//=============================================================================
// ST10_Flow14_B2Press.scl
// 1:1 CONVERSION FROM TIA PORTAL V18 GRAPH XML
// Generated: 2026-02-02
//=============================================================================

TYPE
    E_STEP_ST10_Flow14_B2Press : (
        STEP_ST10_Flow14_B2Press_S2 := 2,
        STEP_ST10_Flow14_B2Press_MesCheckResult_1 := 309,
        STEP_ST10_Flow14_B2Press_ResultOKData := 145,
        STEP_ST10_Flow14_B2Press_B_PressFitting_01CylinderToHP_1 := 140,
        STEP_ST10_Flow14_B2Press_Process_FInish := 237,
        STEP_ST10_Flow14_B2Press_ShaftAndRingOK := 16,
        STEP_ST10_Flow14_B2Press_PutRing := 127,
        STEP_ST10_Flow14_B2Press_PressProgram_1 := 20,
        STEP_ST10_Flow14_B2Press_MESOK := 19,
        STEP_ST10_Flow14_B2Press_Wait_robot_finish_task := 131,
        STEP_ST10_Flow14_B2Press_Step15 := 24,
        STEP_ST10_Flow14_B2Press_Wait__robot_finish_task_1 := 134,
        STEP_ST10_Flow14_B2Press_Status_Alarm := 118,
        STEP_ST10_Flow14_B2Press_StartCycle := 141,
        STEP_ST10_Flow14_B2Press_PressProgram := 8,
        STEP_ST10_Flow14_B2Press_Step400 := 400,
        STEP_ST10_Flow14_B2Press_NGCount := 404,
        STEP_ST10_Flow14_B2Press_RobotLeavePress_Area := 115,
        STEP_ST10_Flow14_B2Press_Part_Check := 239,
        STEP_ST10_Flow14_B2Press_Bypass := 316,
        STEP_ST10_Flow14_B2Press_PartStatus_1 := 137,
        STEP_ST10_Flow14_B2Press_B_PressFitting_01GripperCylinderToHP := 116,
        STEP_ST10_Flow14_B2Press_Bypass_1 := 319,
        STEP_ST10_Flow14_B2Press_Wait_robot_in_safety_area := 133,
        STEP_ST10_Flow14_B2Press_Request_robot_putShaft := 112,
        STEP_ST10_Flow14_B2Press_Prepare_MES_CheckData := 305,
        STEP_ST10_Flow14_B2Press_MesCheckIn_1 := 314,
        STEP_ST10_Flow14_B2Press_PartCheck := 238,
        STEP_ST10_Flow14_B2Press_Step313 := 317,
        STEP_ST10_Flow14_B2Press_Pressing := 200,
        STEP_ST10_Flow14_B2Press_Request_robot_pick := 408,
        STEP_ST10_Flow14_B2Press_ProcessStart := 100,
        STEP_ST10_Flow14_B2Press_MES := 18,
        STEP_ST10_Flow14_B2Press_CheckPressGripStatus := 15,
        STEP_ST10_Flow14_B2Press_MES_1NG := 25,
        STEP_ST10_Flow14_B2Press_CheckPressSensor := 138,
        STEP_ST10_Flow14_B2Press_PressHoming := 9,
        STEP_ST10_Flow14_B2Press_F14_Initial := 1,
        STEP_ST10_Flow14_B2Press_DataMove := 132,
        STEP_ST10_Flow14_B2Press_MES_Check_NG_3 := 318,
        STEP_ST10_Flow14_B2Press_MESOverTime_1 := 312,
        STEP_ST10_Flow14_B2Press_ProcessFInish_1 := 143,
        STEP_ST10_Flow14_B2Press_ShaftOK := 125,
        STEP_ST10_Flow14_B2Press_ProcessFinish := 403,
        STEP_ST10_Flow14_B2Press_PressHoming_1 := 21,
        STEP_ST10_Flow14_B2Press_ResetMesCheckRequest := 301,
        STEP_ST10_Flow14_B2Press_B_PressFitting_01CylinderToHP := 120,
        STEP_ST10_Flow14_B2Press_CheckPressProgram := 139,
        STEP_ST10_Flow14_B2Press_CheckPressResult := 144,
        STEP_ST10_Flow14_B2Press_OKCount := 402,
        STEP_ST10_Flow14_B2Press_PressHoming_ := 13,
        STEP_ST10_Flow14_B2Press_MES_Result := 500,
        STEP_ST10_Flow14_B2Press_ProcessFinsh := 605,
        STEP_ST10_Flow14_B2Press_Request_robot_putRing := 113,
        STEP_ST10_Flow14_B2Press_MES_Check_Finish := 515,
        STEP_ST10_Flow14_B2Press_WaitPressFinish := 201,
        STEP_ST10_Flow14_B2Press_S3 := 3,
        STEP_ST10_Flow14_B2Press_CheckFinish_1 := 315,
        STEP_ST10_Flow14_B2Press_PressReady__1 := 22,
        STEP_ST10_Flow14_B2Press_B_PressFitting_01GripperCylinderToWP := 119,
        STEP_ST10_Flow14_B2Press_DataClear := 604,
        STEP_ST10_Flow14_B2Press_Step314 := 320,
        STEP_ST10_Flow14_B2Press_MES_Check_NG_2 := 313,
        STEP_ST10_Flow14_B2Press_ProductCheckAlarm := 240,
        STEP_ST10_Flow14_B2Press_CheckRingExist := 117,
        STEP_ST10_Flow14_B2Press_ProcessStart_CTStart := 104,
        STEP_ST10_Flow14_B2Press_RobotPick := 600,
        STEP_ST10_Flow14_B2Press_ResetMesUnloadRequest_1 := 302,
        STEP_ST10_Flow14_B2Press_CheckPressReady := 208,
        STEP_ST10_Flow14_B2Press_ProductCheckAlarm_1 := 241,
        STEP_ST10_Flow14_B2Press_StatusAlarm := 126,
        STEP_ST10_Flow14_B2Press_ResultNGData := 146,
        STEP_ST10_Flow14_B2Press_MESOverTime := 321,
        STEP_ST10_Flow14_B2Press_JudgeStatus := 401,
        STEP_ST10_Flow14_B2Press_PressHoming__1 := 23,
        STEP_ST10_Flow14_B2Press_PressReady_ := 12,
        STEP_ST10_Flow14_B2Press_Prepare_MES_CheckData_1 := 307,
        STEP_ST10_Flow14_B2Press_Normal_mode := 103,
        STEP_ST10_Flow14_B2Press_Step147 := 147,
        STEP_ST10_Flow14_B2Press_S5_MESInitial := 5,
        STEP_ST10_Flow14_B2Press_NoPart := 129,
        STEP_ST10_Flow14_B2Press_Wait__robot_finish_task := 130,
        STEP_ST10_Flow14_B2Press_PartStatus := 123,
        STEP_ST10_Flow14_B2Press_Press_NG := 17,
        STEP_ST10_Flow14_B2Press_CheckMachineStatus := 102,
        STEP_ST10_Flow14_B2Press_ok_1 := 322,
        STEP_ST10_Flow14_B2Press_Step14 := 14,
        STEP_ST10_Flow14_B2Press_Determine_product_status := 101,
        STEP_ST10_Flow14_B2Press_MES_Result_OK_1 := 405,
        STEP_ST10_Flow14_B2Press_MES__Check___In := 150,
        STEP_ST10_Flow14_B2Press_RobotLeavePressArea := 121,
        STEP_ST10_Flow14_B2Press_S10_InitialFinish := 10,
        STEP_ST10_Flow14_B2Press_S4 := 4,
        STEP_ST10_Flow14_B2Press_ResetPressStart := 142,
    ) INT := 1;
END_TYPE

CONST
    STEP_ST10_Flow14_B2Press_S2 := 2;
    STEP_ST10_Flow14_B2Press_MesCheckResult_1 := 309;
    STEP_ST10_Flow14_B2Press_ResultOKData := 145;
    STEP_ST10_Flow14_B2Press_B_PressFitting_01CylinderToHP_1 := 140;
    STEP_ST10_Flow14_B2Press_Process_FInish := 237;
    STEP_ST10_Flow14_B2Press_ShaftAndRingOK := 16;
    STEP_ST10_Flow14_B2Press_PutRing := 127;
    STEP_ST10_Flow14_B2Press_PressProgram_1 := 20;
    STEP_ST10_Flow14_B2Press_MESOK := 19;
    STEP_ST10_Flow14_B2Press_Wait_robot_finish_task := 131;
    STEP_ST10_Flow14_B2Press_Step15 := 24;
    STEP_ST10_Flow14_B2Press_Wait__robot_finish_task_1 := 134;
    STEP_ST10_Flow14_B2Press_Status_Alarm := 118;
    STEP_ST10_Flow14_B2Press_StartCycle := 141;
    STEP_ST10_Flow14_B2Press_PressProgram := 8;
    STEP_ST10_Flow14_B2Press_Step400 := 400;
    STEP_ST10_Flow14_B2Press_NGCount := 404;
    STEP_ST10_Flow14_B2Press_RobotLeavePress_Area := 115;
    STEP_ST10_Flow14_B2Press_Part_Check := 239;
    STEP_ST10_Flow14_B2Press_Bypass := 316;
    STEP_ST10_Flow14_B2Press_PartStatus_1 := 137;
    STEP_ST10_Flow14_B2Press_B_PressFitting_01GripperCylinderToHP := 116;
    STEP_ST10_Flow14_B2Press_Bypass_1 := 319;
    STEP_ST10_Flow14_B2Press_Wait_robot_in_safety_area := 133;
    STEP_ST10_Flow14_B2Press_Request_robot_putShaft := 112;
    STEP_ST10_Flow14_B2Press_Prepare_MES_CheckData := 305;
    STEP_ST10_Flow14_B2Press_MesCheckIn_1 := 314;
    STEP_ST10_Flow14_B2Press_PartCheck := 238;
    STEP_ST10_Flow14_B2Press_Step313 := 317;
    STEP_ST10_Flow14_B2Press_Pressing := 200;
    STEP_ST10_Flow14_B2Press_Request_robot_pick := 408;
    STEP_ST10_Flow14_B2Press_ProcessStart := 100;
    STEP_ST10_Flow14_B2Press_MES := 18;
    STEP_ST10_Flow14_B2Press_CheckPressGripStatus := 15;
    STEP_ST10_Flow14_B2Press_MES_1NG := 25;
    STEP_ST10_Flow14_B2Press_CheckPressSensor := 138;
    STEP_ST10_Flow14_B2Press_PressHoming := 9;
    STEP_ST10_Flow14_B2Press_F14_Initial := 1;
    STEP_ST10_Flow14_B2Press_DataMove := 132;
    STEP_ST10_Flow14_B2Press_MES_Check_NG_3 := 318;
    STEP_ST10_Flow14_B2Press_MESOverTime_1 := 312;
    STEP_ST10_Flow14_B2Press_ProcessFInish_1 := 143;
    STEP_ST10_Flow14_B2Press_ShaftOK := 125;
    STEP_ST10_Flow14_B2Press_ProcessFinish := 403;
    STEP_ST10_Flow14_B2Press_PressHoming_1 := 21;
    STEP_ST10_Flow14_B2Press_ResetMesCheckRequest := 301;
    STEP_ST10_Flow14_B2Press_B_PressFitting_01CylinderToHP := 120;
    STEP_ST10_Flow14_B2Press_CheckPressProgram := 139;
    STEP_ST10_Flow14_B2Press_CheckPressResult := 144;
    STEP_ST10_Flow14_B2Press_OKCount := 402;
    STEP_ST10_Flow14_B2Press_PressHoming_ := 13;
    STEP_ST10_Flow14_B2Press_MES_Result := 500;
    STEP_ST10_Flow14_B2Press_ProcessFinsh := 605;
    STEP_ST10_Flow14_B2Press_Request_robot_putRing := 113;
    STEP_ST10_Flow14_B2Press_MES_Check_Finish := 515;
    STEP_ST10_Flow14_B2Press_WaitPressFinish := 201;
    STEP_ST10_Flow14_B2Press_S3 := 3;
    STEP_ST10_Flow14_B2Press_CheckFinish_1 := 315;
    STEP_ST10_Flow14_B2Press_PressReady__1 := 22;
    STEP_ST10_Flow14_B2Press_B_PressFitting_01GripperCylinderToWP := 119;
    STEP_ST10_Flow14_B2Press_DataClear := 604;
    STEP_ST10_Flow14_B2Press_Step314 := 320;
    STEP_ST10_Flow14_B2Press_MES_Check_NG_2 := 313;
    STEP_ST10_Flow14_B2Press_ProductCheckAlarm := 240;
    STEP_ST10_Flow14_B2Press_CheckRingExist := 117;
    STEP_ST10_Flow14_B2Press_ProcessStart_CTStart := 104;
    STEP_ST10_Flow14_B2Press_RobotPick := 600;
    STEP_ST10_Flow14_B2Press_ResetMesUnloadRequest_1 := 302;
    STEP_ST10_Flow14_B2Press_CheckPressReady := 208;
    STEP_ST10_Flow14_B2Press_ProductCheckAlarm_1 := 241;
    STEP_ST10_Flow14_B2Press_StatusAlarm := 126;
    STEP_ST10_Flow14_B2Press_ResultNGData := 146;
    STEP_ST10_Flow14_B2Press_MESOverTime := 321;
    STEP_ST10_Flow14_B2Press_JudgeStatus := 401;
    STEP_ST10_Flow14_B2Press_PressHoming__1 := 23;
    STEP_ST10_Flow14_B2Press_PressReady_ := 12;
    STEP_ST10_Flow14_B2Press_Prepare_MES_CheckData_1 := 307;
    STEP_ST10_Flow14_B2Press_Normal_mode := 103;
    STEP_ST10_Flow14_B2Press_Step147 := 147;
    STEP_ST10_Flow14_B2Press_S5_MESInitial := 5;
    STEP_ST10_Flow14_B2Press_NoPart := 129;
    STEP_ST10_Flow14_B2Press_Wait__robot_finish_task := 130;
    STEP_ST10_Flow14_B2Press_PartStatus := 123;
    STEP_ST10_Flow14_B2Press_Press_NG := 17;
    STEP_ST10_Flow14_B2Press_CheckMachineStatus := 102;
    STEP_ST10_Flow14_B2Press_ok_1 := 322;
    STEP_ST10_Flow14_B2Press_Step14 := 14;
    STEP_ST10_Flow14_B2Press_Determine_product_status := 101;
    STEP_ST10_Flow14_B2Press_MES_Result_OK_1 := 405;
    STEP_ST10_Flow14_B2Press_MES__Check___In := 150;
    STEP_ST10_Flow14_B2Press_RobotLeavePressArea := 121;
    STEP_ST10_Flow14_B2Press_S10_InitialFinish := 10;
    STEP_ST10_Flow14_B2Press_S4 := 4;
    STEP_ST10_Flow14_B2Press_ResetPressStart := 142;
END_CONST

FUNCTION_BLOCK "ST10_Flow14_B2Press_1to1"
{ S7_Optimized_Access := 'TRUE' }
VERSION : 1.0

VAR_INPUT
    iSysInface : "RCS_SysComInterface_V1";
END_VAR

VAR_IN_OUT
    ioPM_Inface : "RCS_PMInterface_V1";
    ioStatus : Int;
END_VAR

VAR_OUTPUT
    oAlarmID : Int;
END_VAR

VAR
    State : INT := 1;
    act_InitialRun : Bool;
    act_InitialOK : Bool;
    act_WaitRunning : Bool;
    act_Running : Bool;
    act_ProcessComplete : Bool;
    act_ProcessStart : Bool;
    act_UnPause : Bool;
    bError : Bool;
    wErrorID : Word;
END_VAR

BEGIN
    //======================================================================
    // STATE MACHINE - Inline Transition Conditions
    //======================================================================

    CASE #State OF

        // ===========================================
        // STEP 2: S2
        // ===========================================
        STEP_ST10_Flow14_B2Press_S2:
            // No actions in XML

            // Transition to next step: 309
            IF TRUE THEN  // Sequential transition - review XML for actual condition
                #State := STEP_ST10_Flow14_B2Press_MesCheckResult_1;
            END_IF;

        // ===========================================
        // STEP 309: MesCheckResult_1
        // ===========================================
        STEP_ST10_Flow14_B2Press_MesCheckResult_1:
            // Action Qualifier=N
            // Token: "PLCtoMES"."PLC.Unload_Station7DataSaveReq"
            "PLCtoMES"."PLC.Unload_Station7DataSaveReq";

            // Transition to next step: 145
            IF TRUE THEN  // Sequential transition - review XML for actual condition
                #State := STEP_ST10_Flow14_B2Press_ResultOKData;
            END_IF;

        // ===========================================
        // STEP 145: ResultOKData
        // ===========================================
        STEP_ST10_Flow14_B2Press_ResultOKData:
            // Action Qualifier=N
            // Token: "AutoProcessData".B_Press2.PartStatus := 480
            "AutoProcessData".B_Press2.PartStatus := 480;

            // Transition to next step: 140
            IF TRUE THEN  // Sequential transition - review XML for actual condition
                #State := STEP_ST10_Flow14_B2Press_B_PressFitting_01CylinderToHP_1;
            END_IF;

        // ===========================================
        // STEP 140: B-PressFitting-01CylinderToHP_1
        // ===========================================
        STEP_ST10_Flow14_B2Press_B_PressFitting_01CylinderToHP_1:
            // Action Qualifier=S
            // Token: "ST10Cylinder".Cy[8].Inout.AutoGoHome
            "ST10Cylinder".Cy[8].Inout.AutoGoHome := TRUE;
            // Action Qualifier=R
            // Token: "ST10Cylinder".Cy[8].Inout.AutoGoWork
            "ST10Cylinder".Cy[8].Inout.AutoGoWork := FALSE;

            // Transition to next step: 237
            IF TRUE THEN  // Sequential transition - review XML for actual condition
                #State := STEP_ST10_Flow14_B2Press_Process_FInish;
            END_IF;

        // ===========================================
        // STEP 237: Process FInish
        // ===========================================
        STEP_ST10_Flow14_B2Press_Process_FInish:
            // No actions in XML

            // Transition to next step: 16
            IF TRUE THEN  // Sequential transition - review XML for actual condition
                #State := STEP_ST10_Flow14_B2Press_ShaftAndRingOK;
            END_IF;

        // ===========================================
        // STEP 16: ShaftAndRingOK
        // ===========================================
        STEP_ST10_Flow14_B2Press_ShaftAndRingOK:
            // No actions in XML

            // Transition to next step: 127
            IF TRUE THEN  // Sequential transition - review XML for actual condition
                #State := STEP_ST10_Flow14_B2Press_PutRing;
            END_IF;

        // ===========================================
        // STEP 127: PutRing
        // ===========================================
        STEP_ST10_Flow14_B2Press_PutRing:
            // No actions in XML

            // Transition to next step: 20
            IF TRUE THEN  // Sequential transition - review XML for actual condition
                #State := STEP_ST10_Flow14_B2Press_PressProgram_1;
            END_IF;

        // ===========================================
        // STEP 20: PressProgram_1
        // ===========================================
        STEP_ST10_Flow14_B2Press_PressProgram_1:
            // Action Qualifier=N
            // Token: "DB_maXYmosNC2".ProgNo := 1
            "DB_maXYmosNC2".ProgNo := 1;

            // Transition to next step: 19
            IF TRUE THEN  // Sequential transition - review XML for actual condition
                #State := STEP_ST10_Flow14_B2Press_MESOK;
            END_IF;

        // ===========================================
        // STEP 19: MESOK
        // ===========================================
        STEP_ST10_Flow14_B2Press_MESOK:
            // No actions in XML

            // Transition to next step: 131
            IF TRUE THEN  // Sequential transition - review XML for actual condition
                #State := STEP_ST10_Flow14_B2Press_Wait_robot_finish_task;
            END_IF;

        // ===========================================
        // STEP 131: Wait robot finish task
        // ===========================================
        STEP_ST10_Flow14_B2Press_Wait_robot_finish_task:
            // No actions in XML

            // Transition to next step: 24
            IF TRUE THEN  // Sequential transition - review XML for actual condition
                #State := STEP_ST10_Flow14_B2Press_Step15;
            END_IF;

        // ===========================================
        // STEP 24: Step15
        // ===========================================
        STEP_ST10_Flow14_B2Press_Step15:
            // No actions in XML

            // Transition to next step: 134
            IF TRUE THEN  // Sequential transition - review XML for actual condition
                #State := STEP_ST10_Flow14_B2Press_Wait__robot_finish_task_1;
            END_IF;

        // ===========================================
        // STEP 134: Wait  robot finish task_1
        // ===========================================
        STEP_ST10_Flow14_B2Press_Wait__robot_finish_task_1:
            // No actions in XML

            // Transition to next step: 118
            IF TRUE THEN  // Sequential transition - review XML for actual condition
                #State := STEP_ST10_Flow14_B2Press_Status_Alarm;
            END_IF;

        // ===========================================
        // STEP 118: Status Alarm
        // ===========================================
        STEP_ST10_Flow14_B2Press_Status_Alarm:
            // Action Qualifier=S
            // Token: "ST10_DeviceError".B.B2Press.StatusError
            "ST10_DeviceError".B.B2Press.StatusError := TRUE;

            // Transition to next step: 141
            IF TRUE THEN  // Sequential transition - review XML for actual condition
                #State := STEP_ST10_Flow14_B2Press_StartCycle;
            END_IF;

        // ===========================================
        // STEP 141: StartCycle
        // ===========================================
        STEP_ST10_Flow14_B2Press_StartCycle:
            // Action Qualifier=S
            // Token: "DB_maXYmosNC2".StartCycle
            "DB_maXYmosNC2".StartCycle := TRUE;

            // Transition to next step: 8
            IF TRUE THEN  // Sequential transition - review XML for actual condition
                #State := STEP_ST10_Flow14_B2Press_PressProgram;
            END_IF;

        // ===========================================
        // STEP 8: PressProgram
        // ===========================================
        STEP_ST10_Flow14_B2Press_PressProgram:
            // Action Qualifier=N
            // Token: "DB_maXYmosNC2".ProgNo := 1
            "DB_maXYmosNC2".ProgNo := 1;

            // Transition to next step: 400
            IF TRUE THEN  // Sequential transition - review XML for actual condition
                #State := STEP_ST10_Flow14_B2Press_Step400;
            END_IF;

        // ===========================================
        // STEP 400: Step400
        // ===========================================
        STEP_ST10_Flow14_B2Press_Step400:
            // No actions in XML

            // Transition to next step: 404
            IF TRUE THEN  // Sequential transition - review XML for actual condition
                #State := STEP_ST10_Flow14_B2Press_NGCount;
            END_IF;

        // ===========================================
        // STEP 404: NGCount
        // ===========================================
        STEP_ST10_Flow14_B2Press_NGCount:
            // Action Qualifier=N
            // Token: #ioPM_Inface.ProcessResult := #ioStatus
            #ioPM_Inface.ProcessResult := #ioStatus;

            // Transition to next step: 115
            IF TRUE THEN  // Sequential transition - review XML for actual condition
                #State := STEP_ST10_Flow14_B2Press_RobotLeavePress_Area;
            END_IF;

        // ===========================================
        // STEP 115: RobotLeavePress Area
        // ===========================================
        STEP_ST10_Flow14_B2Press_RobotLeavePress_Area:
            // No actions in XML

            // Transition to next step: 239
            IF TRUE THEN  // Sequential transition - review XML for actual condition
                #State := STEP_ST10_Flow14_B2Press_Part_Check;
            END_IF;

        // ===========================================
        // STEP 239: Part Check
        // ===========================================
        STEP_ST10_Flow14_B2Press_Part_Check:
            // No actions in XML

            // Transition to next step: 316
            IF TRUE THEN  // Sequential transition - review XML for actual condition
                #State := STEP_ST10_Flow14_B2Press_Bypass;
            END_IF;

        // ===========================================
        // STEP 316: Bypass
        // ===========================================
        STEP_ST10_Flow14_B2Press_Bypass:
            // No actions in XML

            // Transition to next step: 137
            IF TRUE THEN  // Sequential transition - review XML for actual condition
                #State := STEP_ST10_Flow14_B2Press_PartStatus_1;
            END_IF;

        // ===========================================
        // STEP 137: PartStatus_1
        // ===========================================
        STEP_ST10_Flow14_B2Press_PartStatus_1:
            // Action Qualifier=N
            // Token: "AutoProcessData".B_Press2.PartStatus := 450
            "AutoProcessData".B_Press2.PartStatus := 450;

            // Transition to next step: 116
            IF TRUE THEN  // Sequential transition - review XML for actual condition
                #State := STEP_ST10_Flow14_B2Press_B_PressFitting_01GripperCylinderToHP;
            END_IF;

        // ===========================================
        // STEP 116: B-PressFitting-01GripperCylinderToHP
        // ===========================================
        STEP_ST10_Flow14_B2Press_B_PressFitting_01GripperCylinderToHP:
            // Action Qualifier=S
            // Token: "ST10Cylinder".Cy[7].Inout.AutoGoHome
            "ST10Cylinder".Cy[7].Inout.AutoGoHome := TRUE;
            // Action Qualifier=R
            // Token: "ST10Cylinder".Cy[7].Inout.AutoGoWork
            "ST10Cylinder".Cy[7].Inout.AutoGoWork := FALSE;

            // Transition to next step: 319
            IF TRUE THEN  // Sequential transition - review XML for actual condition
                #State := STEP_ST10_Flow14_B2Press_Bypass_1;
            END_IF;

        // ===========================================
        // STEP 319: Bypass_1
        // ===========================================
        STEP_ST10_Flow14_B2Press_Bypass_1:
            // No actions in XML

            // Transition to next step: 133
            IF TRUE THEN  // Sequential transition - review XML for actual condition
                #State := STEP_ST10_Flow14_B2Press_Wait_robot_in_safety_area;
            END_IF;

        // ===========================================
        // STEP 133: Wait robot in safety area
        // ===========================================
        STEP_ST10_Flow14_B2Press_Wait_robot_in_safety_area:
            // No actions in XML

            // Transition to next step: 112
            IF TRUE THEN  // Sequential transition - review XML for actual condition
                #State := STEP_ST10_Flow14_B2Press_Request_robot_putShaft;
            END_IF;

        // ===========================================
        // STEP 112: Request robot putShaft
        // ===========================================
        STEP_ST10_Flow14_B2Press_Request_robot_putShaft:
            // Action Qualifier=N
            // Token: "AutoProcessControl".B_Press_2.Robot2PutPrimit
            "AutoProcessControl".B_Press_2.Robot2PutPrimit;

            // Transition to next step: 305
            IF TRUE THEN  // Sequential transition - review XML for actual condition
                #State := STEP_ST10_Flow14_B2Press_Prepare_MES_CheckData;
            END_IF;

        // ===========================================
        // STEP 305: Prepare MES CheckData
        // ===========================================
        STEP_ST10_Flow14_B2Press_Prepare_MES_CheckData:
            // No actions in XML

            // Transition to next step: 314
            IF TRUE THEN  // Sequential transition - review XML for actual condition
                #State := STEP_ST10_Flow14_B2Press_MesCheckIn_1;
            END_IF;

        // ===========================================
        // STEP 314: MesCheckIn_1
        // ===========================================
        STEP_ST10_Flow14_B2Press_MesCheckIn_1:
            // Action Qualifier=N
            // Token: "PLCtoMES"."PLC.Load_Station7ChickInReq"
            "PLCtoMES"."PLC.Load_Station7ChickInReq";

            // Transition to next step: 238
            IF TRUE THEN  // Sequential transition - review XML for actual condition
                #State := STEP_ST10_Flow14_B2Press_PartCheck;
            END_IF;

        // ===========================================
        // STEP 238: PartCheck
        // ===========================================
        STEP_ST10_Flow14_B2Press_PartCheck:
            // No actions in XML

            // Transition to next step: 317
            IF TRUE THEN  // Sequential transition - review XML for actual condition
                #State := STEP_ST10_Flow14_B2Press_Step313;
            END_IF;

        // ===========================================
        // STEP 317: Step313
        // ===========================================
        STEP_ST10_Flow14_B2Press_Step313:
            // No actions in XML

            // Transition to next step: 200
            IF TRUE THEN  // Sequential transition - review XML for actual condition
                #State := STEP_ST10_Flow14_B2Press_Pressing;
            END_IF;

        // ===========================================
        // STEP 200: Pressing
        // ===========================================
        STEP_ST10_Flow14_B2Press_Pressing:
            // No actions in XML

            // Transition to next step: 408
            IF TRUE THEN  // Sequential transition - review XML for actual condition
                #State := STEP_ST10_Flow14_B2Press_Request_robot_pick;
            END_IF;

        // ===========================================
        // STEP 408: Request robot pick
        // ===========================================
        STEP_ST10_Flow14_B2Press_Request_robot_pick:
            // Action Qualifier=N
            // Token: "AutoProcessControl".B_Press_2.Robot3PickPrimit
            "AutoProcessControl".B_Press_2.Robot3PickPrimit;

            // Transition to next step: 100
            IF TRUE THEN  // Sequential transition - review XML for actual condition
                #State := STEP_ST10_Flow14_B2Press_ProcessStart;
            END_IF;

        // ===========================================
        // STEP 100: ProcessStart
        // ===========================================
        STEP_ST10_Flow14_B2Press_ProcessStart:
            // Action Qualifier=R
            // Token: #ioPM_Inface.InitialRun
            #ioPM_Inface.InitialRun := FALSE;
            // Action Qualifier=R
            // Token: #ioPM_Inface.ProcessComplete
            #ioPM_Inface.ProcessComplete := FALSE;
            // Action Qualifier=S
            // Token: #ioPM_Inface.ProcessStart
            #ioPM_Inface.ProcessStart := TRUE;
            // Action Qualifier=S
            // Token: #ioPM_Inface.InitialOK
            #ioPM_Inface.InitialOK := TRUE;
            // Action Qualifier=S
            // Token: #ioPM_Inface.WaitRunning
            #ioPM_Inface.WaitRunning := TRUE;
            // Action Qualifier=N, Event="S1"
            // Token: #ioPM_Inface.ProcessResult := 0
            #ioPM_Inface.ProcessResult := 0;
            // Action Qualifier=R
            // Token: "ST10_GeneralData".FlowControl_Handshake[14].Start
            "ST10_GeneralData".FlowControl_Handshake[14].Start := FALSE;
            // Action Qualifier=R
            // Token: "ST10_GeneralData".FlowControl_Handshake[14].Done
            "ST10_GeneralData".FlowControl_Handshake[14].Done := FALSE;

            // Transition to next step: 18
            IF TRUE THEN  // Sequential transition - review XML for actual condition
                #State := STEP_ST10_Flow14_B2Press_MES;
            END_IF;

        // ===========================================
        // STEP 18: MES
        // ===========================================
        STEP_ST10_Flow14_B2Press_MES:
            // No actions in XML

            // Transition to next step: 15
            IF TRUE THEN  // Sequential transition - review XML for actual condition
                #State := STEP_ST10_Flow14_B2Press_CheckPressGripStatus;
            END_IF;

        // ===========================================
        // STEP 15: CheckPressGripStatus
        // ===========================================
        STEP_ST10_Flow14_B2Press_CheckPressGripStatus:
            // No actions in XML

            // Transition to next step: 25
            IF TRUE THEN  // Sequential transition - review XML for actual condition
                #State := STEP_ST10_Flow14_B2Press_MES_1NG;
            END_IF;

        // ===========================================
        // STEP 25: MES_1NG
        // ===========================================
        STEP_ST10_Flow14_B2Press_MES_1NG:
            // No actions in XML

            // Transition to next step: 138
            IF TRUE THEN  // Sequential transition - review XML for actual condition
                #State := STEP_ST10_Flow14_B2Press_CheckPressSensor;
            END_IF;

        // ===========================================
        // STEP 138: CheckPressSensor
        // ===========================================
        STEP_ST10_Flow14_B2Press_CheckPressSensor:
            // No actions in XML

            // Transition to next step: 9
            IF TRUE THEN  // Sequential transition - review XML for actual condition
                #State := STEP_ST10_Flow14_B2Press_PressHoming;
            END_IF;

        // ===========================================
        // STEP 9: PressHoming
        // ===========================================
        STEP_ST10_Flow14_B2Press_PressHoming:
            // Action Qualifier=N
            // Token: "DB_maXYmosNC2".Homing
            "DB_maXYmosNC2".Homing;

            // Transition to next step: 1
            IF TRUE THEN  // Sequential transition - review XML for actual condition
                #State := STEP_ST10_Flow14_B2Press_F14_Initial;
            END_IF;

        // ===========================================
        // STEP 1: F14_Initial
        // ===========================================
        STEP_ST10_Flow14_B2Press_F14_Initial:
            // Action Qualifier=S
            // Token: #ioPM_Inface.InitialRun
            #ioPM_Inface.InitialRun := TRUE;
            // Action Qualifier=R
            // Token: #ioPM_Inface.InitialOK
            #ioPM_Inface.InitialOK := FALSE;
            // Action Qualifier=R
            // Token: #ioPM_Inface.WaitRunning
            #ioPM_Inface.WaitRunning := FALSE;
            // Action Qualifier=R
            // Token: #ioPM_Inface.Running
            #ioPM_Inface.Running := FALSE;
            // Action Qualifier=R
            // Token: #ioPM_Inface.ProcessComplete
            #ioPM_Inface.ProcessComplete := FALSE;
            // Action Qualifier=R
            // Token: #ioPM_Inface.UnPause
            #ioPM_Inface.UnPause := FALSE;
            // Action Qualifier=R
            // Token: "Station_Sys".Cmd.Calibration
            "Station_Sys".Cmd.Calibration := FALSE;
            // Action Qualifier=R
            // Token: "Station_Sys".Cmd.ChangeOver
            "Station_Sys".Cmd.ChangeOver := FALSE;
            // Action Qualifier=N
            // Token: //"ST350_Sys".Cmd.DryRun
            //"ST350_Sys".Cmd.DryRun;
            // Action Qualifier=R
            // Token: "Station_Sys".Cmd.Reserve
            "Station_Sys".Cmd.Reserve := FALSE;
            // Action Qualifier=R
            // Token: "Station_Sys".Cmd.OneCycle
            "Station_Sys".Cmd.OneCycle := FALSE;
            // Action Qualifier=R
            // Token: "DB_maXYmosNC2".StartCycle
            "DB_maXYmosNC2".StartCycle := FALSE;
            // Action Qualifier=R
            // Token: "DB_maXYmosNC2".StartCycle
            "DB_maXYmosNC2".StartCycle := FALSE;
            // Action Qualifier=R
            // Token: #ioPM_Inface.ProcessStart
            #ioPM_Inface.ProcessStart := FALSE;
            // Action Qualifier=R
            // Token: "AutoProcessControl".B_Press_2.Robot3PickPrimit
            "AutoProcessControl".B_Press_2.Robot3PickPrimit := FALSE;
            // Action Qualifier=R
            // Token: "AutoProcessControl".B_Press_2.Robot3PutRingPrimit
            "AutoProcessControl".B_Press_2.Robot3PutRingPrimit := FALSE;
            // Action Qualifier=R
            // Token: "AutoProcessControl".B_Press_2.Robot2PutPrimit
            "AutoProcessControl".B_Press_2.Robot2PutPrimit := FALSE;

            // Transition to next step: 132
            IF TRUE THEN  // Sequential transition - review XML for actual condition
                #State := STEP_ST10_Flow14_B2Press_DataMove;
            END_IF;

        // ===========================================
        // STEP 132: DataMove
        // ===========================================
        STEP_ST10_Flow14_B2Press_DataMove:
            // No actions in XML

            // Transition to next step: 318
            IF TRUE THEN  // Sequential transition - review XML for actual condition
                #State := STEP_ST10_Flow14_B2Press_MES_Check_NG_3;
            END_IF;

        // ===========================================
        // STEP 318: MES Check NG_3
        // ===========================================
        STEP_ST10_Flow14_B2Press_MES_Check_NG_3:
            // Action Qualifier=N
            // Token: "AutoProcessData".B_Press2.PartStatus := 452
            "AutoProcessData".B_Press2.PartStatus := 452;

            // Transition to next step: 312
            IF TRUE THEN  // Sequential transition - review XML for actual condition
                #State := STEP_ST10_Flow14_B2Press_MESOverTime_1;
            END_IF;

        // ===========================================
        // STEP 312: MESOverTime_1
        // ===========================================
        STEP_ST10_Flow14_B2Press_MESOverTime_1:
            // Action Qualifier=S
            // Token: "ST10_DeviceError".MES_Error.CheckInCompOverTime_7
            "ST10_DeviceError".MES_Error.CheckInCompOverTime_7 := TRUE;

            // Transition to next step: 143
            IF TRUE THEN  // Sequential transition - review XML for actual condition
                #State := STEP_ST10_Flow14_B2Press_ProcessFInish_1;
            END_IF;

        // ===========================================
        // STEP 143: ProcessFInish 1
        // ===========================================
        STEP_ST10_Flow14_B2Press_ProcessFInish_1:
            // No actions in XML

            // Transition to next step: 125
            IF TRUE THEN  // Sequential transition - review XML for actual condition
                #State := STEP_ST10_Flow14_B2Press_ShaftOK;
            END_IF;

        // ===========================================
        // STEP 125: ShaftOK
        // ===========================================
        STEP_ST10_Flow14_B2Press_ShaftOK:
            // No actions in XML

            // Transition to next step: 403
            IF TRUE THEN  // Sequential transition - review XML for actual condition
                #State := STEP_ST10_Flow14_B2Press_ProcessFinish;
            END_IF;

        // ===========================================
        // STEP 403: ProcessFinish
        // ===========================================
        STEP_ST10_Flow14_B2Press_ProcessFinish:
            // No actions in XML

            // Transition to next step: 21
            IF TRUE THEN  // Sequential transition - review XML for actual condition
                #State := STEP_ST10_Flow14_B2Press_PressHoming_1;
            END_IF;

        // ===========================================
        // STEP 21: PressHoming_1
        // ===========================================
        STEP_ST10_Flow14_B2Press_PressHoming_1:
            // Action Qualifier=N
            // Token: "DB_maXYmosNC2".Homing
            "DB_maXYmosNC2".Homing;

            // Transition to next step: 301
            IF TRUE THEN  // Sequential transition - review XML for actual condition
                #State := STEP_ST10_Flow14_B2Press_ResetMesCheckRequest;
            END_IF;

        // ===========================================
        // STEP 301: ResetMesCheckRequest
        // ===========================================
        STEP_ST10_Flow14_B2Press_ResetMesCheckRequest:
            // Action Qualifier=R
            // Token: "PLCtoMES"."PLC.Load_Station7ChickInReq"
            "PLCtoMES"."PLC.Load_Station7ChickInReq" := FALSE;
            // Action Qualifier=R
            // Token: "MEStoPLC"."MES.Load_Station7PartOK"
            "MEStoPLC"."MES.Load_Station7PartOK" := FALSE;
            // Action Qualifier=R
            // Token: "MEStoPLC"."MES.Load_Station7PartNG"
            "MEStoPLC"."MES.Load_Station7PartNG" := FALSE;
            // Action Qualifier=R
            // Token: "MEStoPLC"."MES.Load_Station7ReqMesDone"
            "MEStoPLC"."MES.Load_Station7ReqMesDone" := FALSE;

            // Transition to next step: 120
            IF TRUE THEN  // Sequential transition - review XML for actual condition
                #State := STEP_ST10_Flow14_B2Press_B_PressFitting_01CylinderToHP;
            END_IF;

        // ===========================================
        // STEP 120: B-PressFitting-01CylinderToHP
        // ===========================================
        STEP_ST10_Flow14_B2Press_B_PressFitting_01CylinderToHP:
            // Action Qualifier=S
            // Token: "ST10Cylinder".Cy[8].Inout.AutoGoHome
            "ST10Cylinder".Cy[8].Inout.AutoGoHome := TRUE;
            // Action Qualifier=R
            // Token: "ST10Cylinder".Cy[8].Inout.AutoGoWork
            "ST10Cylinder".Cy[8].Inout.AutoGoWork := FALSE;

            // Transition to next step: 139
            IF TRUE THEN  // Sequential transition - review XML for actual condition
                #State := STEP_ST10_Flow14_B2Press_CheckPressProgram;
            END_IF;

        // ===========================================
        // STEP 139: CheckPressProgram
        // ===========================================
        STEP_ST10_Flow14_B2Press_CheckPressProgram:
            // Action Qualifier=N
            // Token: "AutoProcessData".B_Press2.Press2Program := "DB_maXYmosNC2".InputMessages.StatusBits.MP
            "AutoProcessData".B_Press2.Press2Program := "DB_maXYmosNC2".InputMessages.StatusBits.MP;

            // Transition to next step: 144
            IF TRUE THEN  // Sequential transition - review XML for actual condition
                #State := STEP_ST10_Flow14_B2Press_CheckPressResult;
            END_IF;

        // ===========================================
        // STEP 144: CheckPressResult
        // ===========================================
        STEP_ST10_Flow14_B2Press_CheckPressResult:
            // No actions in XML

            // Transition to next step: 402
            IF TRUE THEN  // Sequential transition - review XML for actual condition
                #State := STEP_ST10_Flow14_B2Press_OKCount;
            END_IF;

        // ===========================================
        // STEP 402: OKCount
        // ===========================================
        STEP_ST10_Flow14_B2Press_OKCount:
            // Action Qualifier=N
            // Token: #ioPM_Inface.ProcessResult := 400
            #ioPM_Inface.ProcessResult := 400;

            // Transition to next step: 13
            IF TRUE THEN  // Sequential transition - review XML for actual condition
                #State := STEP_ST10_Flow14_B2Press_PressHoming_;
            END_IF;

        // ===========================================
        // STEP 13: PressHoming?
        // ===========================================
        STEP_ST10_Flow14_B2Press_PressHoming_:
            // No actions in XML

            // Transition to next step: 500
            IF TRUE THEN  // Sequential transition - review XML for actual condition
                #State := STEP_ST10_Flow14_B2Press_MES_Result;
            END_IF;

        // ===========================================
        // STEP 500: MES Result
        // ===========================================
        STEP_ST10_Flow14_B2Press_MES_Result:
            // No actions in XML

            // Transition to next step: 605
            IF TRUE THEN  // Sequential transition - review XML for actual condition
                #State := STEP_ST10_Flow14_B2Press_ProcessFinsh;
            END_IF;

        // ===========================================
        // STEP 605: ProcessFinsh
        // ===========================================
        STEP_ST10_Flow14_B2Press_ProcessFinsh:
            // Action Qualifier=S
            // Token: #ioPM_Inface.ProcessComplete
            #ioPM_Inface.ProcessComplete := TRUE;
            // Action Qualifier=R
            // Token: #ioPM_Inface.ProcessStart
            #ioPM_Inface.ProcessStart := FALSE;

            // Transition to next step: 113
            IF TRUE THEN  // Sequential transition - review XML for actual condition
                #State := STEP_ST10_Flow14_B2Press_Request_robot_putRing;
            END_IF;

        // ===========================================
        // STEP 113: Request robot putRing
        // ===========================================
        STEP_ST10_Flow14_B2Press_Request_robot_putRing:
            // Action Qualifier=N
            // Token: "AutoProcessControl".B_Press_2.Robot3PutRingPrimit
            "AutoProcessControl".B_Press_2.Robot3PutRingPrimit;

            // Transition to next step: 515
            IF TRUE THEN  // Sequential transition - review XML for actual condition
                #State := STEP_ST10_Flow14_B2Press_MES_Check_Finish;
            END_IF;

        // ===========================================
        // STEP 515: MES Check Finish
        // ===========================================
        STEP_ST10_Flow14_B2Press_MES_Check_Finish:
            // No actions in XML

            // Transition to next step: 201
            IF TRUE THEN  // Sequential transition - review XML for actual condition
                #State := STEP_ST10_Flow14_B2Press_WaitPressFinish;
            END_IF;

        // ===========================================
        // STEP 201: WaitPressFinish
        // ===========================================
        STEP_ST10_Flow14_B2Press_WaitPressFinish:
            // No actions in XML

            // Transition to next step: 3
            IF TRUE THEN  // Sequential transition - review XML for actual condition
                #State := STEP_ST10_Flow14_B2Press_S3;
            END_IF;

        // ===========================================
        // STEP 3: S3
        // ===========================================
        STEP_ST10_Flow14_B2Press_S3:
            // No actions in XML

            // Transition to next step: 315
            IF TRUE THEN  // Sequential transition - review XML for actual condition
                #State := STEP_ST10_Flow14_B2Press_CheckFinish_1;
            END_IF;

        // ===========================================
        // STEP 315: CheckFinish_1
        // ===========================================
        STEP_ST10_Flow14_B2Press_CheckFinish_1:
            // No actions in XML

            // Transition to next step: 22
            IF TRUE THEN  // Sequential transition - review XML for actual condition
                #State := STEP_ST10_Flow14_B2Press_PressReady__1;
            END_IF;

        // ===========================================
        // STEP 22: PressReady?_1
        // ===========================================
        STEP_ST10_Flow14_B2Press_PressReady__1:
            // No actions in XML

            // Transition to next step: 119
            IF TRUE THEN  // Sequential transition - review XML for actual condition
                #State := STEP_ST10_Flow14_B2Press_B_PressFitting_01GripperCylinderToWP;
            END_IF;

        // ===========================================
        // STEP 119: B-PressFitting-01GripperCylinderToWP
        // ===========================================
        STEP_ST10_Flow14_B2Press_B_PressFitting_01GripperCylinderToWP:
            // Action Qualifier=R
            // Token: "ST10Cylinder".Cy[7].Inout.AutoGoHome
            "ST10Cylinder".Cy[7].Inout.AutoGoHome := FALSE;
            // Action Qualifier=S
            // Token: "ST10Cylinder".Cy[7].Inout.AutoGoWork
            "ST10Cylinder".Cy[7].Inout.AutoGoWork := TRUE;

            // Transition to next step: 604
            IF TRUE THEN  // Sequential transition - review XML for actual condition
                #State := STEP_ST10_Flow14_B2Press_DataClear;
            END_IF;

        // ===========================================
        // STEP 604: DataClear
        // ===========================================
        STEP_ST10_Flow14_B2Press_DataClear:
            // Action Qualifier=N, Event="S1"
            // Token: #ioPM_Inface.ProcessResult := 0
            #ioPM_Inface.ProcessResult := 0;
            // Action Qualifier=N, Event="S1"
            // Token: #ioStatus := 0
            #ioStatus := 0;

            // Transition to next step: 320
            IF TRUE THEN  // Sequential transition - review XML for actual condition
                #State := STEP_ST10_Flow14_B2Press_Step314;
            END_IF;

        // ===========================================
        // STEP 320: Step314
        // ===========================================
        STEP_ST10_Flow14_B2Press_Step314:
            // No actions in XML

            // Transition to next step: 313
            IF TRUE THEN  // Sequential transition - review XML for actual condition
                #State := STEP_ST10_Flow14_B2Press_MES_Check_NG_2;
            END_IF;

        // ===========================================
        // STEP 313: MES Check NG_2
        // ===========================================
        STEP_ST10_Flow14_B2Press_MES_Check_NG_2:
            // Action Qualifier=N
            // Token: "AutoProcessData".B_Press2.PartStatus := 451
            "AutoProcessData".B_Press2.PartStatus := 451;

            // Transition to next step: 240
            IF TRUE THEN  // Sequential transition - review XML for actual condition
                #State := STEP_ST10_Flow14_B2Press_ProductCheckAlarm;
            END_IF;

        // ===========================================
        // STEP 240: ProductCheckAlarm
        // ===========================================
        STEP_ST10_Flow14_B2Press_ProductCheckAlarm:
            // Action Qualifier=S
            // Token: "ST10_DeviceError".B.B2Press.ShaftSensorCheckError
            "ST10_DeviceError".B.B2Press.ShaftSensorCheckError := TRUE;

            // Transition to next step: 117
            IF TRUE THEN  // Sequential transition - review XML for actual condition
                #State := STEP_ST10_Flow14_B2Press_CheckRingExist;
            END_IF;

        // ===========================================
        // STEP 117: CheckRingExist
        // ===========================================
        STEP_ST10_Flow14_B2Press_CheckRingExist:
            // No actions in XML

            // Transition to next step: 104
            IF TRUE THEN  // Sequential transition - review XML for actual condition
                #State := STEP_ST10_Flow14_B2Press_ProcessStart_CTStart;
            END_IF;

        // ===========================================
        // STEP 104: ProcessStart,CTStart
        // ===========================================
        STEP_ST10_Flow14_B2Press_ProcessStart_CTStart:
            // No actions in XML

            // Transition to next step: 600
            IF TRUE THEN  // Sequential transition - review XML for actual condition
                #State := STEP_ST10_Flow14_B2Press_RobotPick;
            END_IF;

        // ===========================================
        // STEP 600: RobotPick
        // ===========================================
        STEP_ST10_Flow14_B2Press_RobotPick:
            // No actions in XML

            // Transition to next step: 302
            IF TRUE THEN  // Sequential transition - review XML for actual condition
                #State := STEP_ST10_Flow14_B2Press_ResetMesUnloadRequest_1;
            END_IF;

        // ===========================================
        // STEP 302: ResetMesUnloadRequest_1
        // ===========================================
        STEP_ST10_Flow14_B2Press_ResetMesUnloadRequest_1:
            // Action Qualifier=R
            // Token: "PLCtoMES"."PLC.Unload_Station7DataSaveReq"
            "PLCtoMES"."PLC.Unload_Station7DataSaveReq" := FALSE;
            // Action Qualifier=R
            // Token: "MEStoPLC"."MES.Unload_ResultsStored7OK"
            "MEStoPLC"."MES.Unload_ResultsStored7OK" := FALSE;
            // Action Qualifier=R
            // Token: "MEStoPLC"."MES.Unload_ResultsStored7NG"
            "MEStoPLC"."MES.Unload_ResultsStored7NG" := FALSE;
            // Action Qualifier=R
            // Token: "MEStoPLC"."MES.Unload_ResultsStored7ReqMesDone"
            "MEStoPLC"."MES.Unload_ResultsStored7ReqMesDone" := FALSE;

            // Transition to next step: 208
            IF TRUE THEN  // Sequential transition - review XML for actual condition
                #State := STEP_ST10_Flow14_B2Press_CheckPressReady;
            END_IF;

        // ===========================================
        // STEP 208: CheckPressReady
        // ===========================================
        STEP_ST10_Flow14_B2Press_CheckPressReady:
            // Action Qualifier=R
            // Token: "DB_maXYmosNC2".StartCycle
            "DB_maXYmosNC2".StartCycle := FALSE;

            // Transition to next step: 241
            IF TRUE THEN  // Sequential transition - review XML for actual condition
                #State := STEP_ST10_Flow14_B2Press_ProductCheckAlarm_1;
            END_IF;

        // ===========================================
        // STEP 241: ProductCheckAlarm_1
        // ===========================================
        STEP_ST10_Flow14_B2Press_ProductCheckAlarm_1:
            // Action Qualifier=S
            // Token: "ST10_DeviceError".B.B2Press.RingSensorCheckError
            "ST10_DeviceError".B.B2Press.RingSensorCheckError := TRUE;

            // Transition to next step: 126
            IF TRUE THEN  // Sequential transition - review XML for actual condition
                #State := STEP_ST10_Flow14_B2Press_StatusAlarm;
            END_IF;

        // ===========================================
        // STEP 126: StatusAlarm
        // ===========================================
        STEP_ST10_Flow14_B2Press_StatusAlarm:
            // Action Qualifier=S
            // Token: "ST10_DeviceError".B.B2Press.StatusError
            "ST10_DeviceError".B.B2Press.StatusError := TRUE;

            // Transition to next step: 146
            IF TRUE THEN  // Sequential transition - review XML for actual condition
                #State := STEP_ST10_Flow14_B2Press_ResultNGData;
            END_IF;

        // ===========================================
        // STEP 146: ResultNGData
        // ===========================================
        STEP_ST10_Flow14_B2Press_ResultNGData:
            // Action Qualifier=N
            // Token: "AutoProcessData".B_Press2.PartStatus := 455
            "AutoProcessData".B_Press2.PartStatus := 455;

            // Transition to next step: 321
            IF TRUE THEN  // Sequential transition - review XML for actual condition
                #State := STEP_ST10_Flow14_B2Press_MESOverTime;
            END_IF;

        // ===========================================
        // STEP 321: MESOverTime
        // ===========================================
        STEP_ST10_Flow14_B2Press_MESOverTime:
            // Action Qualifier=S
            // Token: "ST10_DeviceError".MES_Error.CheckInResultOverTime_7
            "ST10_DeviceError".MES_Error.CheckInResultOverTime_7 := TRUE;

            // Transition to next step: 401
            IF TRUE THEN  // Sequential transition - review XML for actual condition
                #State := STEP_ST10_Flow14_B2Press_JudgeStatus;
            END_IF;

        // ===========================================
        // STEP 401: JudgeStatus
        // ===========================================
        STEP_ST10_Flow14_B2Press_JudgeStatus:
            // Action Qualifier=N
            // Token: #ioPM_Inface.ProcessResult := 0
            #ioPM_Inface.ProcessResult := 0;

            // Transition to next step: 23
            IF TRUE THEN  // Sequential transition - review XML for actual condition
                #State := STEP_ST10_Flow14_B2Press_PressHoming__1;
            END_IF;

        // ===========================================
        // STEP 23: PressHoming?_1
        // ===========================================
        STEP_ST10_Flow14_B2Press_PressHoming__1:
            // No actions in XML

            // Transition to next step: 12
            IF TRUE THEN  // Sequential transition - review XML for actual condition
                #State := STEP_ST10_Flow14_B2Press_PressReady_;
            END_IF;

        // ===========================================
        // STEP 12: PressReady?
        // ===========================================
        STEP_ST10_Flow14_B2Press_PressReady_:
            // No actions in XML

            // Transition to next step: 307
            IF TRUE THEN  // Sequential transition - review XML for actual condition
                #State := STEP_ST10_Flow14_B2Press_Prepare_MES_CheckData_1;
            END_IF;

        // ===========================================
        // STEP 307: Prepare MES CheckData_1
        // ===========================================
        STEP_ST10_Flow14_B2Press_Prepare_MES_CheckData_1:
            // No actions in XML

            // Transition to next step: 103
            IF TRUE THEN  // Sequential transition - review XML for actual condition
                #State := STEP_ST10_Flow14_B2Press_Normal_mode;
            END_IF;

        // ===========================================
        // STEP 103: Normal mode
        // ===========================================
        STEP_ST10_Flow14_B2Press_Normal_mode:
            // No actions in XML

            // Transition to next step: 147
            IF TRUE THEN  // Sequential transition - review XML for actual condition
                #State := STEP_ST10_Flow14_B2Press_Step147;
            END_IF;

        // ===========================================
        // STEP 147: Step147
        // ===========================================
        STEP_ST10_Flow14_B2Press_Step147:
            // No actions in XML

            // Transition to next step: 5
            IF TRUE THEN  // Sequential transition - review XML for actual condition
                #State := STEP_ST10_Flow14_B2Press_S5_MESInitial;
            END_IF;

        // ===========================================
        // STEP 5: S5_MESInitial
        // ===========================================
        STEP_ST10_Flow14_B2Press_S5_MESInitial:
            // No actions in XML

            // Transition to next step: 129
            IF TRUE THEN  // Sequential transition - review XML for actual condition
                #State := STEP_ST10_Flow14_B2Press_NoPart;
            END_IF;

        // ===========================================
        // STEP 129: NoPart
        // ===========================================
        STEP_ST10_Flow14_B2Press_NoPart:
            // No actions in XML

            // Transition to next step: 130
            IF TRUE THEN  // Sequential transition - review XML for actual condition
                #State := STEP_ST10_Flow14_B2Press_Wait__robot_finish_task;
            END_IF;

        // ===========================================
        // STEP 130: Wait  robot finish task
        // ===========================================
        STEP_ST10_Flow14_B2Press_Wait__robot_finish_task:
            // No actions in XML

            // Transition to next step: 123
            IF TRUE THEN  // Sequential transition - review XML for actual condition
                #State := STEP_ST10_Flow14_B2Press_PartStatus;
            END_IF;

        // ===========================================
        // STEP 123: PartStatus
        // ===========================================
        STEP_ST10_Flow14_B2Press_PartStatus:
            // No actions in XML

            // Transition to next step: 17
            IF TRUE THEN  // Sequential transition - review XML for actual condition
                #State := STEP_ST10_Flow14_B2Press_Press_NG;
            END_IF;

        // ===========================================
        // STEP 17: Press NG
        // ===========================================
        STEP_ST10_Flow14_B2Press_Press_NG:
            // No actions in XML

            // Transition to next step: 102
            IF TRUE THEN  // Sequential transition - review XML for actual condition
                #State := STEP_ST10_Flow14_B2Press_CheckMachineStatus;
            END_IF;

        // ===========================================
        // STEP 102: CheckMachineStatus
        // ===========================================
        STEP_ST10_Flow14_B2Press_CheckMachineStatus:
            // No actions in XML

            // Transition to next step: 322
            IF TRUE THEN  // Sequential transition - review XML for actual condition
                #State := STEP_ST10_Flow14_B2Press_ok_1;
            END_IF;

        // ===========================================
        // STEP 322: ok_1
        // ===========================================
        STEP_ST10_Flow14_B2Press_ok_1:
            // Action Qualifier=N
            // Token: "AutoProcessData".B_Press2.PartStatus := 499
            "AutoProcessData".B_Press2.PartStatus := 499;

            // Transition to next step: 14
            IF TRUE THEN  // Sequential transition - review XML for actual condition
                #State := STEP_ST10_Flow14_B2Press_Step14;
            END_IF;

        // ===========================================
        // STEP 14: Step14
        // ===========================================
        STEP_ST10_Flow14_B2Press_Step14:
            // No actions in XML

            // Transition to next step: 101
            IF TRUE THEN  // Sequential transition - review XML for actual condition
                #State := STEP_ST10_Flow14_B2Press_Determine_product_status;
            END_IF;

        // ===========================================
        // STEP 101: Determine product status
        // ===========================================
        STEP_ST10_Flow14_B2Press_Determine_product_status:
            // Action Qualifier=N
            // Token: "MES_CHeck_DB".Station_7.CheckStep := 0
            "MES_CHeck_DB".Station_7.CheckStep := 0;
            // Action Qualifier=N
            // Token: "MES_CHeck_DB".Station_7.ResultStep := 0
            "MES_CHeck_DB".Station_7.ResultStep := 0;

            // Transition to next step: 405
            IF TRUE THEN  // Sequential transition - review XML for actual condition
                #State := STEP_ST10_Flow14_B2Press_MES_Result_OK_1;
            END_IF;

        // ===========================================
        // STEP 405: MES Result OK_1
        // ===========================================
        STEP_ST10_Flow14_B2Press_MES_Result_OK_1:
            // Action Qualifier=N
            // Token: "AutoProcessData".B_Press2.PartStatus := 499
            "AutoProcessData".B_Press2.PartStatus := 499;

            // Transition to next step: 150
            IF TRUE THEN  // Sequential transition - review XML for actual condition
                #State := STEP_ST10_Flow14_B2Press_MES__Check___In;
            END_IF;

        // ===========================================
        // STEP 150: MES  Check   In
        // ===========================================
        STEP_ST10_Flow14_B2Press_MES__Check___In:
            // No actions in XML

            // Transition to next step: 121
            IF TRUE THEN  // Sequential transition - review XML for actual condition
                #State := STEP_ST10_Flow14_B2Press_RobotLeavePressArea;
            END_IF;

        // ===========================================
        // STEP 121: RobotLeavePressArea
        // ===========================================
        STEP_ST10_Flow14_B2Press_RobotLeavePressArea:
            // No actions in XML

            // Transition to next step: 10
            IF TRUE THEN  // Sequential transition - review XML for actual condition
                #State := STEP_ST10_Flow14_B2Press_S10_InitialFinish;
            END_IF;

        // ===========================================
        // STEP 10: S10_InitialFinish
        // ===========================================
        STEP_ST10_Flow14_B2Press_S10_InitialFinish:
            // Action Qualifier=S
            // Token: #ioPM_Inface.InitialOK
            #ioPM_Inface.InitialOK := TRUE;

            // Transition to next step: 4
            IF TRUE THEN  // Sequential transition - review XML for actual condition
                #State := STEP_ST10_Flow14_B2Press_S4;
            END_IF;

        // ===========================================
        // STEP 4: S4
        // ===========================================
        STEP_ST10_Flow14_B2Press_S4:
            // No actions in XML

            // Transition to next step: 142
            IF TRUE THEN  // Sequential transition - review XML for actual condition
                #State := STEP_ST10_Flow14_B2Press_ResetPressStart;
            END_IF;

        // ===========================================
        // STEP 142: ResetPressStart
        // ===========================================
        STEP_ST10_Flow14_B2Press_ResetPressStart:
            // Action Qualifier=R
            // Token: "DB_maXYmosNC2".StartCycle
            "DB_maXYmosNC2".StartCycle := FALSE;

    END_CASE;

    // UPDATE ioPM_Inface
    #ioPM_Inface.InitialRun := #act_InitialRun;
    #ioPM_Inface.InitialOK := #act_InitialOK;
    #ioPM_Inface.WaitRunning := #act_WaitRunning;
    #ioPM_Inface.Running := #act_Running;
    #ioPM_Inface.ProcessComplete := #act_ProcessComplete;
    #ioPM_Inface.ProcessStart := #act_ProcessStart;
    #ioPM_Inface.UnPause := #act_UnPause;

    // ERROR HANDLING
    IF #bError THEN
        #ioStatus := 900;
        #oAlarmID := INT_TO_WORD(#wErrorID);
    ELSE
        #ioStatus := 0;
        #oAlarmID := 0;
    END_IF;
END_FUNCTION_BLOCK

//=============================================================================
// END OF FILE
//=============================================================================
